(* POU Выборка значения из массива/Get_Speed_ARRAY_Number, ST *)
FUNCTION Get_Speed_ARRAY_Number : BYTE
VAR_INPUT
	Volume_now:DINT;
END_VAR
VAR
	i:BYTE:=1;
	j,ArraySize:BYTE:=12;
	med:BYTE;
END_VAR
(* Функция в качестве аргумента принимает, давление надува в мВольтах, а возвращает номер элемента массива, соответствующего этому количеству оборотов *)


(* Делим массив каждый раз пополам, проверяя где находится искомый элемент, пока границы массива не сойдутся*)

WHILE i<>j  DO
	med:=(i+j)/2;
	IF Volume_now > p.Speed_table[med] THEN
		i:=med+1;
	ELSE
		j:=med;
	END_IF
END_WHILE


Get_Speed_ARRAY_Number :=i;							(* Номер , когда границы сошлись и совпадают с краями массива не нуждается в уточнении *)

(* Уточняем какой элемент массива наиболее сответствует, кол-ву оборотов переданному как элемент функции *)
(* определяем спава или слева от найдено индекса находится ребуемый элемент и в зависмимости от этого действеум *)

IF i=med AND i<>1 THEN
	IF ABS(p.Speed_table[med-1]-Volume_now)<= ABS(p.Speed_table[med]-Volume_now) THEN
		Get_Speed_ARRAY_Number :=med-1;
	ELSE
		Get_Speed_ARRAY_Number :=med;
	END_IF
ELSIF i<>med AND  i<>ArraySize THEN
	IF ABS(p.Speed_table[med+1]-Volume_now)<= ABS(p.Speed_table[med]-Volume_now) THEN
		Get_Speed_ARRAY_Number :=med+1;
	ELSE
		Get_Speed_ARRAY_Number :=med;
	END_IF
END_IF
END_FUNCTION

(* POU Выборка значения из массива/Get_PPS_ARRAY_Number, ST *)
FUNCTION Get_PPS_ARRAY_Number : BYTE
VAR_INPUT
	PPS_now:DINT;
END_VAR
VAR
	i:BYTE:=1;
	j,ArraySize:BYTE:=32;
	med:BYTE;
END_VAR
(* Функция в качестве аргумента принимает, PPS, а возвращает номер элемента массива, соответствующего этому PPS *)

(* Делим массив каждый раз пополам, проверяя где находится искомый элемент, пока границы массива не сойдутся*)

WHILE i<>j  DO
	med:=(i+j)/2;
	IF PPS_now>p.PPS_table[med] THEN
		i:=med+1;
	ELSE
		j:=med;
	END_IF
END_WHILE


Get_PPS_ARRAY_Number :=i;							(* Номер , когда границы сошлись и совпадают с краями массива не нуждается в уточнении *)

(* Уточняем какой элемент массива наиболее сответствует, кол-ву оборотов переданному как элемент функции *)
(* определяем спава или слева от найдено индекса находится ребуемый элемент и в зависмимости от этого действеум *)

IF i=med AND i<>1 THEN
	IF ABS(p.PPS_table[med-1]-PPS_now)<= ABS(p.RPM_table[med]-PPS_now) THEN
		Get_PPS_ARRAY_Number :=med-1;
	ELSE
		Get_PPS_ARRAY_Number :=med;
	END_IF
ELSIF i<>med AND  i<>ArraySize THEN
	IF ABS(p.PPS_table[med+1]-PPS_now)<= ABS(p.PPS_table[med]-PPS_now) THEN
		Get_PPS_ARRAY_Number :=med+1;
	ELSE
		Get_PPS_ARRAY_Number :=med;
	END_IF
END_IF
END_FUNCTION

(* POU Ввод данных/Get_Turbo, ST *)
PROGRAM Get_Turbo
VAR
	s16_Return      : INT;
   fb_InGetValue   : FB_x_in_get_value;
END_VAR
fb_InGetValue(ou16_Channel:=X_IN_21, os32_Value=>Turbo_pressure, os16_Status=>s16_Return);
END_PROGRAM

(* POU Ввод данных/Get_Key, ST *)
PROGRAM Get_Key
VAR
	s16_Return      : INT;
   fb_InGetValue   : FB_x_in_get_value;

	DF_switch	:DINT;
	DF_flag		:BOOL;

END_VAR
fb_InGetValue(ou16_Channel:=X_IN_12, os32_Value=>DF_switch, os16_Status=>s16_Return);

IF DF_switch=0 THEN					(* Если конпока изменения режима работы ECU нажата, то...*)
	IF DF_flag THEN					(* Первый ли цикл когда она нажата ? *)
		DF_flag:=FALSE;				(*Выставляем флажок, для  игнорирования этой ветви, до тех пор пока кнопка не изменит своего положения *)
		IF Flag_ECU_ON THEN			(* Включаем или выключаем газодизельный режим ECU*)
			Flag_ECU_ON:=FALSE;
		ELSE
			Flag_ECU_ON:=TRUE;
			Count_min_reductor_press:=0; (* При переключении режимов начать отчет времени когда далвение было минимальным с 0 *)
		END_IF;
	END_IF
ELSE
	DF_flag:=TRUE;				(* Кнопка была отпущена, устанвкливаем разрешительный флажок для обработки следующего нажатия *)
END_IF
END_PROGRAM

(* POU Ввод данных/Get_Gas_meter, ST *)
PROGRAM Get_Gas_meter
VAR
	s16_Return      : INT;
   fb_InGetValue   : FB_x_in_get_value;
	fb_OutSetValue   : FB_x_out_set_value;

	i: DINT;
END_VAR
(* Считать значениедатчика кол-ва газа *)
fb_InGetValue(ou16_Channel:=X_IN_19, os32_Value=>Gas_meter, os16_Status=>s16_Return);

(* Определить уровень PWM для зажигания LED *)
i:=p.LED_BAR_PWM[Get_Gas_meter_ARRAY_Number(Gas_meter)];

(* Выдать PWM на LED bar *)
fb_OutSetValue(ou16_Channel:=X_OUT_03, os32_Value:=i, os16_Status=>s16_Return);
END_PROGRAM

(* POU Выборка значения из массива/Get_Gas_meter_ARRAY_Number, ST *)
FUNCTION Get_Gas_meter_ARRAY_Number : BYTE
VAR_INPUT
	Gas_meter_now:DINT;
END_VAR
VAR
	i:BYTE:=1;
	j,ArraySize:BYTE:=5;
	med:BYTE;

END_VAR
(* Функция в качестве аргумента принимает, количество оборотов, а возвращает номер элемента массива, соответствующего этому PPS *)


(* Делим массив каждый раз пополам, проверяя где находится искомый элемент, пока границы массива не сойдутся*)

WHILE i<>j  DO
	med:=(i+j)/2;
	IF Gas_meter_now>p.Gas_meter_volume[med] THEN
		i:=med+1;
	ELSE
		j:=med;
	END_IF
END_WHILE


Get_Gas_meter_ARRAY_Number :=i;							(* Номер , когда границы сошлись и совпадают с краями массива не нуждается в уточнении *)

(* Уточняем какой элемент массива наиболее сответствует, кол-ву оборотов переданному как элемент функции *)
(* определяем спава или слева от найдено индекса находится ребуемый элемент и в зависмимости от этого действеум *)

IF i=med AND i<>1 THEN
	IF ABS(p.Gas_meter_volume[med-1]-Gas_meter_now)<= ABS(p.Gas_meter_volume[med]-Gas_meter_now) THEN
		Get_Gas_meter_ARRAY_Number :=med-1;
	ELSE
		Get_Gas_meter_ARRAY_Number :=med;
	END_IF
ELSIF i<>med AND  i<>ArraySize THEN
	IF ABS(p.Gas_meter_volume[med+1]-Gas_meter_now)<= ABS(p.Gas_meter_volume[med]-Gas_meter_now) THEN
		Get_Gas_meter_ARRAY_Number :=med+1;
	ELSE
		Get_Gas_meter_ARRAY_Number :=med;
	END_IF
END_IF
END_FUNCTION

(* POU Ввод данных/Get_Reductor_temp, ST *)
PROGRAM Get_Reductor_temp
VAR
	s16_Return      : INT;
   fb_InGetValue   : FB_x_in_get_value;

	(* Температура редуктора уже в норме, время до следующей проверки пошло *)
	Flag_Err_Reductor_temp: BOOL;
	(* Счетчик циклов до следующей проверки *)
	Count_max_Reductor_temp: WORD;

END_VAR
fb_InGetValue(ou16_Channel:=X_IN_20, os32_Value=>Reductor_temp, os16_Status=>s16_Return);

(* Если температура редуктора превысила допустимую температуру для включения, то следующий
контроль произойдет через некоторое время,что бы избежать дребезга *)

IF Flag_Err_Reductor_temp AND  Count_max_Reductor_temp < Reductor_temp_err_time THEN
	Count_max_reductor_temp:=Count_max_reductor_temp+1;
ELSE
	Count_max_Reductor_temp:=0;
	(* Находится ли температура редуктора в допустимых пределах ? *)
	IF Reductor_temp < p.Reductor_temp_work THEN
		Flag_Err_Reductor_temp:=TRUE;
		Err_Reductor_temp:=TRUE;
	ELSE
		Flag_Err_Reductor_temp:=FALSE;
		Err_Reductor_temp:=FALSE;
	END_IF
END_IF
END_PROGRAM

(* POU Ввод данных/Get_Inj_temp, ST *)
PROGRAM Get_Inj_temp
VAR
	s16_Return      : INT;
   fb_InGetValue   : FB_x_in_get_value;
END_VAR
fb_InGetValue(ou16_Channel:=X_IN_15, os32_Value=>Injector_temp, os16_Status=>s16_Return);

(* Находится ли температура форсунок в допустимых пределах ? *)
(* Если температура форсунок хоть один раз превысила допустимый порог, то снять ошибку можно только перегрузкой *)

IF Injector_temp > p.Inj_temp_max THEN
	Err_inj_temp:=TRUE;
END_IF
END_PROGRAM

(* POU Ввод данных/Get_FUEL_meter, ST *)
PROGRAM Get_FUEL_meter
VAR
	s16_Return      : INT;
   fb_InGetValue   : FB_x_in_get_value;
	fb_OutSetValue   : FB_x_out_set_value;
	q: WORD;
END_VAR
(* Считать значениедатчика кол-ва солярки *)
fb_InGetValue(ou16_Channel:=X_IN_18, os32_Value=>FUEL_meter, os16_Status=>s16_Return);
(*Взять из таблицы физическое згачение объема слоответствующее показанию датчика *)
q:= p.FUEL_meter_liter[ Get_FUEL_meter_ARRAY_Number(FUEL_meter)];
FUEL_volume:=DINT_TO_REAL(FUEL_meter) * WORD_TO_REAL( q );
IF p.FUEL_meter_dat[Get_FUEL_meter_ARRAY_Number(FUEL_meter)] <> 0 THEN
	FUEL_volume:=FUEL_volume/WORD_TO_REAL(p.FUEL_meter_dat[Get_FUEL_meter_ARRAY_Number(FUEL_meter)]);
END_IF
END_PROGRAM

(* POU Выборка значения из массива/Get_FUEL_meter_ARRAY_Number, ST *)
FUNCTION Get_FUEL_meter_ARRAY_Number : BYTE
VAR_INPUT
	FUEL_meter_now:DINT;
END_VAR
VAR
	i:BYTE:=1;
	j,ArraySize:BYTE:=32;
	med:BYTE;

END_VAR
(* Функция в качестве аргумента принимает, количество оборотов, а возвращает номер элемента массива, соответствующего этому PPS *)


(* Делим массив каждый раз пополам, проверяя где находится искомый элемент, пока границы массива не сойдутся*)

WHILE i<>j  DO
	med:=(i+j)/2;
	IF FUEL_meter_now>p.FUEL_meter_dat[med] THEN
		i:=med+1;
	ELSE
		j:=med;
	END_IF
END_WHILE


Get_FUEL_meter_ARRAY_Number :=i;							(* Номер , когда границы сошлись и совпадают с краями массива не нуждается в уточнении *)

(* Уточняем какой элемент массива наиболее сответствует, кол-ву оборотов переданному как элемент функции *)
(* определяем спава или слева от найдено индекса находится ребуемый элемент и в зависмимости от этого действеум *)

IF i=med AND i<>1 THEN
	IF ABS(p.FUEL_meter_dat[med-1]-FUEL_meter_now)<= ABS(p.FUEL_meter_dat[med]-FUEL_meter_now) THEN
		Get_FUEL_meter_ARRAY_Number :=med-1;
	ELSE
		Get_FUEL_meter_ARRAY_Number :=med;
	END_IF
ELSIF i<>med AND  i<>ArraySize THEN
	IF ABS(p.FUEL_meter_dat[med+1]-FUEL_meter_now)<= ABS(p.FUEL_meter_dat[med]-FUEL_meter_now) THEN
		Get_FUEL_meter_ARRAY_Number :=med+1;
	ELSE
		Get_FUEL_meter_ARRAY_Number :=med;
	END_IF
END_IF
END_FUNCTION

(* POU Ввод данных/Get_cPPS, ST *)
PROGRAM Get_cPPS
VAR
	fb_InGetValue   : FB_x_in_get_value;
	s16_Return      : INT;
END_VAR
(* Взяьть реальное значение выдаваемого напряжения эмуляции PPS *)
fb_InGetValue(ou16_Channel:=X_IN_26, os32_Value=>cPPS1_emul, os16_Status=>s16_Return);
END_PROGRAM

(* POU CAN/Send, ST *)
PROGRAM Send
VAR
	s16_Return       		: INT;
	t_Msg             	: T_x_can_msg;
   fb_CanObjSendMsg   	: FB_x_can_obj_send_msg;
	fb_EepRead  			: FB_x_eep_read;
	u16_Crc           	: UINT;
	fb_UtiCalcCrc16   	: FB_x_uti_calc_crc_16;
	CAN_TX_count			:WORD:=10000;				(* Счетчик переданных пакетов по CAN *)

END_VAR
IF Flag_CAN THEN

	IF Flag_CAN_Write THEN
		Flag_CAN_Write:=FALSE;
		t_Msg.t_Id.u32_Id := 16#101;
		t_Msg.t_Id.u8_Xtd := 0;
		t_Msg.u8_Dlc      := 8;				(* Количество передаваемых байт *)
		t_Msg.au8_Data[0] := 1;
		t_Msg.au8_Data[1] := 9;
		t_Msg.au8_Data[2] := 7;
		t_Msg.au8_Data[3] := 2;
		t_Msg.au8_Data[4] := 1;
		t_Msg.au8_Data[5] := 9;
		t_Msg.au8_Data[6] := 7;
		t_Msg.au8_Data[7] := 2;
		fb_CanObjSendMsg(ou32_Handle:=TX, ot_Msg:=t_Msg, os16_Status=>s16_Return);
	END_IF


	IF Flag_CAN_send THEN											(* Первоначальная процедура, выполняется один раз по команде от Питоновской программе *)
		(* Читаем все содержимое энергонезависимой памяти *)
		fb_EepRead(ou32_Address:=0, ou32_Count:=SIZEOF(Can_buffer), opu8_Data:=ADR(Can_buffer), os16_Status=>s16_Return);
		(* Вычисляем CRC16 для массива передаваемых данных *)
		u16_Crc:=16#1D0F;
		fb_UtiCalcCrc16(ou32_Count:=SIZEOF(Can_buffer)-2, opu8_Data:=ADR(Can_buffer), ou16_Crc:=u16_Crc, os16_Status=>s16_Return);
		Can_buffer[SIZEOF(Can_buffer)-1]:=WORD_TO_BYTE(u16_Crc);
		Can_buffer[SIZEOF(Can_buffer)]:=WORD_TO_BYTE(u16_Crc/256);
		CAN_TX_count:=0;
		Flag_CAN_send:=FALSE;


	ELSIF CAN_TX_count <=  (SIZEOF(Can_buffer)-8) THEN						(* Передача основных данных, выполняется 1 раз после хандшейка *)

			(* Постоянная часть передачи *)
			t_Msg.t_Id.u32_Id := 16#101;		(* Адрес пакета *)
			t_Msg.t_Id.u8_Xtd := 0;
			t_Msg.u8_Dlc      := 8;				(* Количество передаваемых байт *)
			t_Msg.au8_Data[0] := Can_buffer[CAN_TX_count+1];
			t_Msg.au8_Data[1] := Can_buffer[CAN_TX_count+2];
			t_Msg.au8_Data[2] := Can_buffer[CAN_TX_count+3];
			t_Msg.au8_Data[3] := Can_buffer[CAN_TX_count+4];
			t_Msg.au8_Data[4] := Can_buffer[CAN_TX_count+5];
			t_Msg.au8_Data[5] := Can_buffer[CAN_TX_count+6];
			t_Msg.au8_Data[6] := Can_buffer[CAN_TX_count+7];
			t_Msg.au8_Data[7] := Can_buffer[CAN_TX_count+8];
			fb_CanObjSendMsg(ou32_Handle:=TX, ot_Msg:=t_Msg, os16_Status=>s16_Return);
			CAN_TX_count:=CAN_TX_count+8;
		END_IF

END_IF
END_PROGRAM

(* POU CAN/Recieve, ST *)
PROGRAM Recieve
VAR
	s16_Return        	: INT;
	r_Msg			         : T_x_can_msg;
	fb_CanObjGetMsg   	: FB_x_can_obj_get_msg;
	fb_EepWrite  			: FB_x_eep_write;

	u16_Crc           	: UINT;
	fb_UtiCalcCrc16   	: FB_x_uti_calc_crc_16;
	i: WORD; (* Счетчик принятых по CAN пакетов в калибровке *)

	crc_given: UINT;
END_VAR
IF Flag_CAN THEN
			(* Что бы при ошибке чтения с CANa , при не изменении значений не произошо ложного срабатывания *)
			r_Msg.au8_Data[0]:=0;r_Msg.au8_Data[1]:=0;r_Msg.au8_Data[2]:=0;r_Msg.au8_Data[3]:=0;r_Msg.au8_Data[4]:=0;
			r_Msg.au8_Data[5]:=0;r_Msg.au8_Data[6]:=0;r_Msg.au8_Data[7]:=0;
			fb_CanObjGetMsg(ou32_Handle:=RX, ot_Msg=>r_Msg, os16_Status=>s16_Return);
			IF s16_Return = C_NO_ERR THEN

					(* Поступил запрос на передачу? *)
					IF	Flag_CAN_recieve=FALSE AND r_Msg.au8_Data[0] = 8 AND r_Msg.au8_Data[1] = 7 AND r_Msg.au8_Data[2] = 6 AND r_Msg.au8_Data[3] = 5 AND
						r_Msg.au8_Data[4] = 4 AND r_Msg.au8_Data[5] = 3 AND r_Msg.au8_Data[6] = 2 AND	r_Msg.au8_Data[7] = 1 THEN
						Flag_CAN_send:=TRUE;
					END_IF

					(* Поступил запрос на прием ? *)
					IF Flag_CAN_recieve = FALSE AND r_Msg.au8_Data[0] = 1 AND r_Msg.au8_Data[1] = 2 AND r_Msg.au8_Data[2] = 3 AND r_Msg.au8_Data[3] = 4 AND
						r_Msg.au8_Data[4] = 5 AND r_Msg.au8_Data[5] = 6 AND r_Msg.au8_Data[6] = 7 AND r_Msg.au8_Data[7] = 8 THEN

									Flag_CAN_recieve:=TRUE;
									i:=1;
					ELSIF i <= SIZEOF(Can_buffer)-7 THEN
											Can_buffer[i]:=r_Msg.au8_Data[0]; Can_buffer[i+1]:=r_Msg.au8_Data[1]; Can_buffer[i+2]:=r_Msg.au8_Data[2]; Can_buffer[i+3]:=r_Msg.au8_Data[3];
											Can_buffer[i+4]:=r_Msg.au8_Data[4]; Can_buffer[i+5]:=r_Msg.au8_Data[5]; Can_buffer[i+6]:=r_Msg.au8_Data[6]; Can_buffer[i+7]:=r_Msg.au8_Data[7];
											i:=i+8;
											IF i=SIZEOF(Can_buffer)+1 THEN
													Flag_CAN_recieve:= FALSE;
													(* Вычисляем CRC16 для массива передаваемых данных *)
													u16_Crc:=16#1D0F;
													fb_UtiCalcCrc16(ou32_Count:=SIZEOF(Can_buffer)-2, opu8_Data:=ADR(Can_buffer), ou16_Crc:=u16_Crc, os16_Status=>s16_Return);
													crc_given:= Can_buffer[SIZEOF(Can_buffer)]*256+Can_buffer[SIZEOF(Can_buffer)-1];
													IF crc_given =  u16_Crc THEN
															fb_EepWrite(ou32_Address:=0, ou32_Count:=SIZEOF(Can_buffer), opu8_Data:=ADR(Can_buffer), os16_Status=>s16_Return);
															Flag_CAN_Write:= TRUE;
													END_IF
											END_IF
					END_IF

			END_IF
END_IF
END_PROGRAM

(* Visualisation CALIBRATION
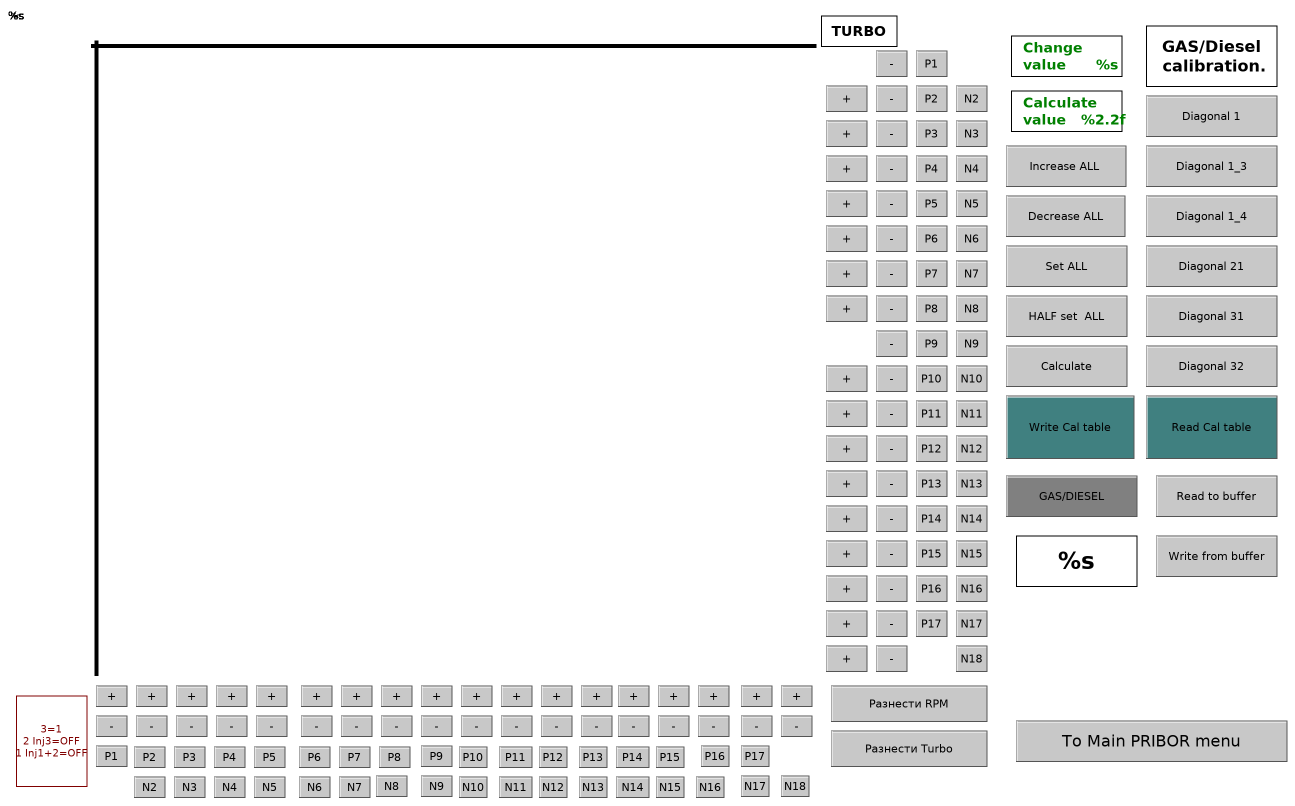
rectangle at (0,0)-(0,0): text "%s"; shows p.RPM_table[INDEX]; editable
rectangle at (0,0)-(0,0): text "%s"; shows p.Turbo_table[1]; editable
rectangle at (0,0)-(0,0): text "%s"; shows p.Turbo_table[2]; editable
rectangle at (0,0)-(0,0): text "%s"; shows p.Turbo_table[3]; editable
rectangle at (0,0)-(0,0): text "%s"; shows p.Turbo_table[4]; editable
rectangle at (0,0)-(0,0): text "%s"; shows p.Turbo_table[5]; editable
rectangle at (0,0)-(0,0): text "%s"; shows p.Turbo_table[6]; editable
rectangle at (0,0)-(0,0): text "%s"; shows p.Turbo_table[7]; editable
rectangle at (0,0)-(0,0): text "%s"; shows p.Turbo_table[8]; editable
rectangle at (0,0)-(0,0): text "%s"; shows p.Turbo_table[9]; editable
rectangle at (0,0)-(0,0): text "%s"; shows p.Turbo_table[10]; editable
rectangle at (0,0)-(0,0): text "%s"; shows p.Turbo_table[11]; editable
rectangle at (0,0)-(0,0): text "%s"; shows p.Turbo_table[12]; editable
rectangle at (0,0)-(0,0): text "%s"; shows p.Turbo_table[13]; editable
rectangle at (0,0)-(0,0): text "%s"; shows p.Turbo_table[14]; editable
rectangle at (0,0)-(0,0): text "%s"; shows p.Turbo_table[15]; editable
rectangle at (0,0)-(0,0): text "%s"; shows p.Turbo_table[16]; editable
rectangle at (0,0)-(0,0): text "%s"; shows p.Turbo_table[17]; editable
rectangle at (0,0)-(0,0): text "%s"; shows p.Turbo_table[18]; editable
button at (990,130)-(1110,171): text "Increase ALL"; taps DFPRS_Change_Cal_Table.ALL_plus
button at (990,180)-(1109,221): text "Decrease ALL"; taps DFPRS_Change_Cal_Table.ALL_minus
button at (1130,380)-(1261,443): text "Read Cal table"; taps DFPRS_Change_Cal_Table.Read_cal
button at (990,380)-(1118,443): text "Write Cal table"; taps DFPRS_Change_Cal_Table.Write_cal
button at (990,230)-(1111,271): text "Set ALL"; taps DFPRS_Change_Cal_Table.Set_ALL
button at (990,280)-(1111,321): text "HALF set  ALL"; taps DFPRS_Change_Cal_Table.HALF_set_ALL
button at (860,35)-(891,61): text "-"; taps DFPRS_Change_Cal_Table.RPM_Flag_minus_1
button at (810,70)-(851,96): text "+"; taps DFPRS_Change_Cal_Table.RPM_Flag_plus_2
button at (860,70)-(891,96): text "-"; taps DFPRS_Change_Cal_Table.RPM_Flag_minus_2
button at (900,70)-(931,96): text "P2"; taps DFPRS_Change_Cal_Table.RPM_Flag_CP_2
button at (810,105)-(851,131): text "+"; taps DFPRS_Change_Cal_Table.RPM_Flag_plus_3
button at (860,105)-(891,131): text "-"; taps DFPRS_Change_Cal_Table.RPM_Flag_minus_3
button at (900,105)-(931,131): text "P3"; taps DFPRS_Change_Cal_Table.RPM_Flag_CP_3
button at (810,140)-(851,166): text "+"; taps DFPRS_Change_Cal_Table.RPM_Flag_plus_4
button at (860,140)-(891,166): text "-"; taps DFPRS_Change_Cal_Table.RPM_Flag_minus_4
button at (900,140)-(931,166): text "P4"; taps DFPRS_Change_Cal_Table.RPM_Flag_CP_4
button at (810,175)-(851,201): text "+"; taps DFPRS_Change_Cal_Table.RPM_Flag_plus_5
button at (860,175)-(891,201): text "-"; taps DFPRS_Change_Cal_Table.RPM_Flag_minus_5
button at (900,175)-(931,201): text "P5"; taps DFPRS_Change_Cal_Table.RPM_Flag_CP_5
button at (810,210)-(851,236): text "+"; taps DFPRS_Change_Cal_Table.RPM_Flag_plus_6
button at (860,210)-(891,236): text "-"; taps DFPRS_Change_Cal_Table.RPM_Flag_minus_6
button at (900,210)-(931,236): text "P6"; taps DFPRS_Change_Cal_Table.RPM_Flag_CP_6
button at (810,245)-(851,271): text "+"; taps DFPRS_Change_Cal_Table.RPM_Flag_plus_7
button at (860,245)-(891,271): text "-"; taps DFPRS_Change_Cal_Table.RPM_Flag_minus_7
button at (900,245)-(931,271): text "P7"; taps DFPRS_Change_Cal_Table.RPM_Flag_CP_7
button at (810,280)-(851,306): text "+"; taps DFPRS_Change_Cal_Table.RPM_Flag_plus_8
button at (860,280)-(891,306): text "-"; taps DFPRS_Change_Cal_Table.RPM_Flag_minus_8
button at (900,280)-(931,306): text "P8"; taps DFPRS_Change_Cal_Table.RPM_Flag_CP_8
button at (80,670)-(111,691): text "+"; taps DFPRS_Change_Cal_Table.Turbo_Flag_plus_1
button at (80,700)-(111,721): text "-"; taps DFPRS_Change_Cal_Table.Turbo_Flag_minus_1
button at (120,670)-(151,691): text "+"; taps DFPRS_Change_Cal_Table.Turbo_Flag_plus_2
button at (120,700)-(151,721): text "-"; taps DFPRS_Change_Cal_Table.Turbo_Flag_minus_2
button at (118,731)-(149,752): text "P2"; taps DFPRS_Change_Cal_Table.Turbo_Flag_CP_2
button at (160,670)-(191,691): text "+"; taps DFPRS_Change_Cal_Table.Turbo_Flag_plus_3
button at (160,700)-(191,721): text "-"; taps DFPRS_Change_Cal_Table.Turbo_Flag_minus_3
button at (158,731)-(189,752): text "P3"; taps DFPRS_Change_Cal_Table.Turbo_Flag_CP_3
button at (200,670)-(231,691): text "+"; taps DFPRS_Change_Cal_Table.Turbo_Flag_plus_4
button at (200,700)-(231,721): text "-"; taps DFPRS_Change_Cal_Table.Turbo_Flag_minus_4
button at (198,731)-(229,752): text "P4"; taps DFPRS_Change_Cal_Table.Turbo_Flag_CP_4
button at (240,670)-(271,691): text "+"; taps DFPRS_Change_Cal_Table.Turbo_Flag_plus_5
button at (240,700)-(271,721): text "-"; taps DFPRS_Change_Cal_Table.Turbo_Flag_minus_5
button at (238,731)-(269,752): text "P5"; taps DFPRS_Change_Cal_Table.Turbo_Flag_CP_5
button at (285,670)-(316,691): text "+"; taps DFPRS_Change_Cal_Table.Turbo_Flag_plus_6
button at (285,700)-(316,721): text "-"; taps DFPRS_Change_Cal_Table.Turbo_Flag_minus_6
button at (283,731)-(314,752): text "P6"; taps DFPRS_Change_Cal_Table.Turbo_Flag_CP_6
button at (325,670)-(356,691): text "+"; taps DFPRS_Change_Cal_Table.Turbo_Flag_plus_7
button at (325,700)-(356,721): text "-"; taps DFPRS_Change_Cal_Table.Turbo_Flag_minus_7
button at (323,731)-(354,752): text "P7"; taps DFPRS_Change_Cal_Table.Turbo_Flag_CP_7
button at (365,670)-(396,691): text "+"; taps DFPRS_Change_Cal_Table.Turbo_Flag_plus_8
button at (365,700)-(396,721): text "-"; taps DFPRS_Change_Cal_Table.Turbo_Flag_minus_8
button at (363,731)-(394,752): text "P8"; taps DFPRS_Change_Cal_Table.Turbo_Flag_CP_8
rounded rectangle at (995,20)-(1106,61): text "Change / value      %s"; shows DFPRS_Change_Cal_Table.Change_volume; editable 0..
rounded rectangle at (1130,10)-(1261,71): text "GAS/Diesel / calibration."
button at (1140,460)-(1261,501): text "Read to buffer"; taps DFPRS_Change_Cal_Table.red_cal2
button at (1140,520)-(1261,561): text "Write from buffer"; taps DFPRS_Change_Cal_Table.Write_cal2
button at (860,315)-(891,341): text "-"; taps DFPRS_Change_Cal_Table.RPM_Flag_minus_9
button at (810,350)-(851,376): text "+"; taps DFPRS_Change_Cal_Table.RPM_Flag_plus_10
button at (860,350)-(891,376): text "-"; taps DFPRS_Change_Cal_Table.RPM_Flag_minus_10
button at (900,350)-(931,376): text "P10"; taps DFPRS_Change_Cal_Table.RPM_Flag_CP_10
button at (810,385)-(851,411): text "+"; taps DFPRS_Change_Cal_Table.RPM_Flag_plus_11
button at (860,385)-(891,411): text "-"; taps DFPRS_Change_Cal_Table.RPM_Flag_minus_11
button at (900,385)-(931,411): text "P11"; taps DFPRS_Change_Cal_Table.RPM_Flag_CP_11
button at (810,420)-(851,446): text "+"; taps DFPRS_Change_Cal_Table.RPM_Flag_plus_12
button at (860,420)-(891,446): text "-"; taps DFPRS_Change_Cal_Table.RPM_Flag_minus_12
button at (900,420)-(931,446): text "P12"; taps DFPRS_Change_Cal_Table.RPM_Flag_CP_12
button at (810,455)-(851,481): text "+"; taps DFPRS_Change_Cal_Table.RPM_Flag_plus_13
button at (860,455)-(891,481): text "-"; taps DFPRS_Change_Cal_Table.RPM_Flag_minus_13
button at (900,455)-(931,481): text "P13"; taps DFPRS_Change_Cal_Table.RPM_Flag_CP_13
button at (900,315)-(931,341): text "P9"; taps DFPRS_Change_Cal_Table.RPM_Flag_CP_9
button at (405,670)-(436,691): text "+"; taps DFPRS_Change_Cal_Table.Turbo_Flag_plus_9
button at (405,700)-(436,721): text "-"; taps DFPRS_Change_Cal_Table.Turbo_Flag_minus_9
button at (445,670)-(476,691): text "+"; taps DFPRS_Change_Cal_Table.Turbo_Flag_plus_10
button at (445,700)-(476,721): text "-"; taps DFPRS_Change_Cal_Table.Turbo_Flag_minus_10
button at (443,731)-(471,752): text "P10"; taps DFPRS_Change_Cal_Table.Turbo_Flag_CP_10
button at (485,670)-(516,691): text "+"; taps DFPRS_Change_Cal_Table.Turbo_Flag_plus_11
button at (485,700)-(516,721): text "-"; taps DFPRS_Change_Cal_Table.Turbo_Flag_minus_11
button at (483,731)-(516,752): text "P11"; taps DFPRS_Change_Cal_Table.Turbo_Flag_CP_11
button at (525,670)-(556,691): text "+"; taps DFPRS_Change_Cal_Table.Turbo_Flag_plus_12
button at (525,700)-(556,721): text "-"; taps DFPRS_Change_Cal_Table.Turbo_Flag_minus_12
button at (523,731)-(551,752): text "P12"; taps DFPRS_Change_Cal_Table.Turbo_Flag_CP_12
button at (565,670)-(596,691): text "+"; taps DFPRS_Change_Cal_Table.Turbo_Flag_plus_13
button at (565,700)-(596,721): text "-"; taps DFPRS_Change_Cal_Table.Turbo_Flag_minus_13
button at (563,731)-(591,752): text "P13"; taps DFPRS_Change_Cal_Table.Turbo_Flag_CP_13
button at (405,730)-(436,751): text "P9"; taps DFPRS_Change_Cal_Table.Turbo_Flag_CP_9
rectangle at (0,680)-(71,771): text "3=1 / 2 Inj3=OFF / 1 Inj1+2=OFF"
button at (990,460)-(1121,501): text "GAS/DIESEL"; toggles DFPRS_Change_Cal_Table.Flag_cal_table_gas
rounded rectangle at (1000,520)-(1121,571): text "%s"; shows DFPRS_Change_Cal_Table.Fuel_type
button at (990,330)-(1111,371): text "Calculate"; taps DFPRS_Change_Cal_Table.Calculate
rounded rectangle at (995,75)-(1106,116): text "Calculate / value   %2.2f"; shows .p.Calculate_volume; editable 0..
button at (1130,80)-(1261,121): text "Diagonal 1"; taps DFPRS_Change_Cal_Table.Diagonal_1
button at (810,490)-(851,516): text "+"; taps DFPRS_Change_Cal_Table.RPM_Flag_plus_14
button at (860,490)-(891,516): text "-"; taps DFPRS_Change_Cal_Table.RPM_Flag_minus_14
button at (900,490)-(931,516): text "P14"; taps DFPRS_Change_Cal_Table.RPM_Flag_CP_14
button at (810,525)-(851,551): text "+"; taps DFPRS_Change_Cal_Table.RPM_Flag_plus_15
button at (860,525)-(891,551): text "-"; taps DFPRS_Change_Cal_Table.RPM_Flag_minus_15
button at (900,525)-(931,551): text "P15"; taps DFPRS_Change_Cal_Table.RPM_Flag_CP_15
button at (810,560)-(851,586): text "+"; taps DFPRS_Change_Cal_Table.RPM_Flag_plus_16
button at (860,560)-(891,586): text "-"; taps DFPRS_Change_Cal_Table.RPM_Flag_minus_16
button at (900,35)-(931,61): text "P1"; taps DFPRS_Change_Cal_Table.RPM_Flag_CP_1
button at (940,70)-(971,96): text "N2"; taps DFPRS_Change_Cal_Table.RPM_Flag_CN_2
button at (940,105)-(971,131): text "N3"; taps DFPRS_Change_Cal_Table.RPM_Flag_CN_3
button at (940,140)-(971,166): text "N4"; taps DFPRS_Change_Cal_Table.RPM_Flag_CN_4
button at (940,175)-(971,201): text "N5"; taps DFPRS_Change_Cal_Table.RPM_Flag_CN_5
button at (940,210)-(971,236): text "N6"; taps DFPRS_Change_Cal_Table.RPM_Flag_CN_6
button at (940,245)-(971,271): text "N7"; taps DFPRS_Change_Cal_Table.RPM_Flag_CN_7
button at (940,280)-(971,306): text "N8"; taps DFPRS_Change_Cal_Table.RPM_Flag_CN_8
button at (940,350)-(971,376): text "N10"; taps DFPRS_Change_Cal_Table.RPM_Flag_CN_10
button at (940,385)-(971,411): text "N11"; taps DFPRS_Change_Cal_Table.RPM_Flag_CN_11
button at (940,420)-(971,446): text "N12"; taps DFPRS_Change_Cal_Table.RPM_Flag_CN_12
button at (940,455)-(971,481): text "N13"; taps DFPRS_Change_Cal_Table.RPM_Flag_CN_13
button at (940,315)-(971,341): text "N9"; taps DFPRS_Change_Cal_Table.RPM_Flag_CN_9
button at (940,490)-(971,516): text "N14"; taps DFPRS_Change_Cal_Table.RPM_Flag_CN_14
button at (940,525)-(971,551): text "N15"; taps DFPRS_Change_Cal_Table.RPM_Flag_CN_15
button at (940,560)-(971,586): text "N16"; taps DFPRS_Change_Cal_Table.RPM_Flag_CN_16
button at (1130,180)-(1261,221): text "Diagonal 1_4"; taps DFPRS_Change_Cal_Table.Diagonal_14
button at (1130,130)-(1261,171): text "Diagonal 1_3"; taps DFPRS_Change_Cal_Table.Diagonal_13
button at (1130,230)-(1261,271): text "Diagonal 21"; taps DFPRS_Change_Cal_Table.Diagonal_21
button at (1130,280)-(1261,321): text "Diagonal 31"; taps DFPRS_Change_Cal_Table.Diagonal_31
button at (1000,705)-(1271,746): text "To Main PRIBOR menu"; opens PLC_VISU
button at (602,670)-(633,691): text "+"; taps DFPRS_Change_Cal_Table.Turbo_Flag_plus_14
button at (602,700)-(633,721): text "-"; taps DFPRS_Change_Cal_Table.Turbo_Flag_minus_14
button at (600,731)-(633,752): text "P14"; taps DFPRS_Change_Cal_Table.Turbo_Flag_CP_14
button at (642,670)-(673,691): text "+"; taps DFPRS_Change_Cal_Table.Turbo_Flag_plus_15
button at (642,700)-(673,721): text "-"; taps DFPRS_Change_Cal_Table.Turbo_Flag_minus_15
button at (640,731)-(668,752): text "P15"; taps DFPRS_Change_Cal_Table.Turbo_Flag_CP_15
button at (682,670)-(713,691): text "+"; taps DFPRS_Change_Cal_Table.Turbo_Flag_plus_16
button at (682,700)-(713,721): text "-"; taps DFPRS_Change_Cal_Table.Turbo_Flag_minus_16
button at (80,730)-(111,751): text "P1"; taps DFPRS_Change_Cal_Table.Turbo_Flag_CP_1
button at (118,761)-(149,782): text "N2"; taps DFPRS_Change_Cal_Table.Turbo_Flag_CN_2
button at (158,761)-(189,782): text "N3"; taps DFPRS_Change_Cal_Table.Turbo_Flag_CN_3
button at (198,761)-(229,782): text "N4"; taps DFPRS_Change_Cal_Table.Turbo_Flag_CN_4
button at (238,761)-(269,782): text "N5"; taps DFPRS_Change_Cal_Table.Turbo_Flag_CN_5
button at (283,761)-(314,782): text "N6"; taps DFPRS_Change_Cal_Table.Turbo_Flag_CN_6
button at (323,761)-(354,782): text "N7"; taps DFPRS_Change_Cal_Table.Turbo_Flag_CN_7
button at (360,760)-(391,781): text "N8"; taps DFPRS_Change_Cal_Table.Turbo_Flag_CN_8
button at (443,761)-(471,782): text "N10"; taps DFPRS_Change_Cal_Table.Turbo_Flag_CN_10
button at (483,761)-(516,782): text "N11"; taps DFPRS_Change_Cal_Table.Turbo_Flag_CN_11
button at (523,761)-(551,782): text "N12"; taps DFPRS_Change_Cal_Table.Turbo_Flag_CN_12
button at (563,761)-(591,782): text "N13"; taps DFPRS_Change_Cal_Table.Turbo_Flag_CN_13
button at (405,760)-(436,781): text "N9"; taps DFPRS_Change_Cal_Table.Turbo_Flag_CN_9
button at (600,761)-(633,782): text "N14"; taps DFPRS_Change_Cal_Table.Turbo_Flag_CN_14
button at (640,761)-(668,782): text "N15"; taps DFPRS_Change_Cal_Table.Turbo_Flag_CN_15
button at (680,761)-(708,782): text "N16"; taps DFPRS_Change_Cal_Table.Turbo_Flag_CN_16
button at (1130,330)-(1261,371): text "Diagonal 32"; taps DFPRS_Change_Cal_Table.Diagonal_32
rectangle at (805,0)-(881,31): text "TURBO"
button at (810,595)-(851,621): text "+"; taps DFPRS_Change_Cal_Table.RPM_Flag_plus_17
button at (860,595)-(891,621): text "-"; taps DFPRS_Change_Cal_Table.RPM_Flag_minus_17
button at (810,630)-(851,656): text "+"; taps DFPRS_Change_Cal_Table.RPM_Flag_plus_18
button at (860,630)-(891,656): text "-"; taps DFPRS_Change_Cal_Table.RPM_Flag_minus_18
button at (725,670)-(756,691): text "+"; taps DFPRS_Change_Cal_Table.Turbo_Flag_plus_17
button at (725,700)-(756,721): text "-"; taps DFPRS_Change_Cal_Table.Turbo_Flag_minus_17
button at (765,670)-(796,691): text "+"; taps DFPRS_Change_Cal_Table.Turbo_Flag_plus_18
button at (765,700)-(796,721): text "-"; taps DFPRS_Change_Cal_Table.Turbo_Flag_minus_18
button at (900,595)-(931,621): text "P17"; taps DFPRS_Change_Cal_Table.RPM_Flag_CP_17
button at (940,595)-(971,621): text "N17"; taps DFPRS_Change_Cal_Table.RPM_Flag_CN_17
button at (940,630)-(971,656): text "N18"; taps DFPRS_Change_Cal_Table.RPM_Flag_CN_18
button at (900,560)-(931,586): text "P16"; taps DFPRS_Change_Cal_Table.RPM_Flag_CP_16
button at (725,730)-(753,751): text "P17"; taps DFPRS_Change_Cal_Table.Turbo_Flag_CP_17
button at (725,760)-(753,781): text "N17"; taps DFPRS_Change_Cal_Table.Turbo_Flag_CN_17
button at (765,760)-(793,781): text "N18"; taps DFPRS_Change_Cal_Table.Turbo_Flag_CN_18
button at (685,730)-(713,751): text "P16"; taps DFPRS_Change_Cal_Table.Turbo_Flag_CP_16
button at (815,670)-(971,706): text "Разнести RPM"; taps DFPRS_Change_Cal_Table.Flag_RPM_raznoska
button at (815,715)-(971,751): text "Разнести Turbo"; taps DFPRS_Change_Cal_Table.Flag_Turbo_raznoska
2 more shapes without text or variables
*)

(* Visualisation Check_parameters/CHECK_CURRENT
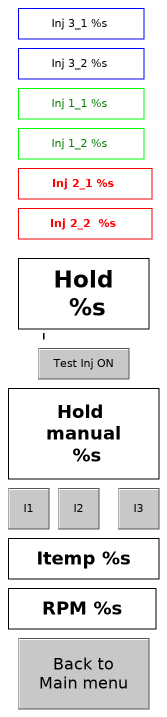
rounded rectangle at (1210,90)-(1336,121): text "Inj 1_1 %s"; shows .s32_Current_Inj1_1/1000
rounded rectangle at (1210,210)-(1344,241): text "Inj 2_2  %s"; shows .s32_Current_Inj2_2/1000
rounded rectangle at (1210,260)-(1341,331): text "Hold / %s"; shows .HOLD_time
rounded rectangle at (1210,10)-(1336,41): text "Inj 3_1 %s"; shows .s32_Current_Inj3_1/1000
rounded rectangle at (1210,130)-(1336,161): text "Inj 1_2 %s"; shows .s32_Current_Inj1_2/1000
rounded rectangle at (1210,170)-(1344,201): text "Inj 2_1 %s"; shows .s32_Current_Inj2_1/1000
rounded rectangle at (1210,50)-(1336,81): text "Inj 3_2 %s"; shows s32_Current_Inj3_2/1000
button at (1230,350)-(1321,381): text "Test Inj ON"; toggles .Flag_test_inj
rectangle at (1200,390)-(1351,481): text "Hold / manual / %s"; shows Act_control.Hold_manual; editable
button at (1200,490)-(1241,531): text "I1"; toggles .Flag_Inj1_ON
button at (1250,490)-(1291,531): text "I2"; toggles .Flag_Inj2_ON
button at (1310,490)-(1351,531): text "I3"; toggles .Flag_Inj3_ON
rounded rectangle at (1200,540)-(1351,581): text "Itemp %s"; shows .Injector_temp
rounded rectangle at (1200,590)-(1348,631): text "RPM %s"; shows .RPM
button at (1210,640)-(1341,711): text "Back to / Main menu"; opens PLC_VISU
1 more shapes without text or variables
1 elements of other kinds (tables, trends, ...) not read
*)

(* Visualisation Check_parameters/CHECK_EGT
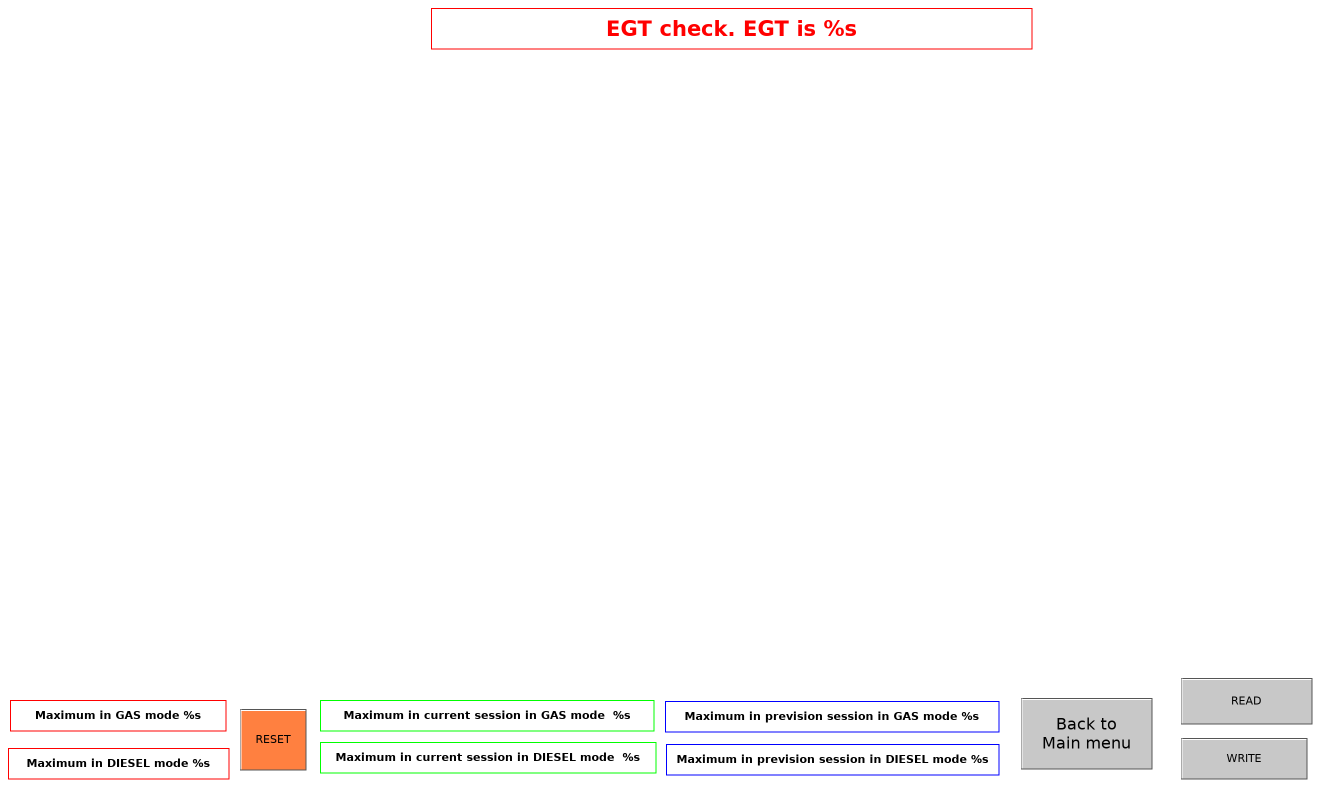
rounded rectangle at (9,702)-(225,733): text "Maximum in GAS mode %s"; shows .a.EGT_max_abs_GAS
rounded rectangle at (7,750)-(228,781): text "Maximum in DIESEL mode %s"; shows .a.EGT_max_abs_DIESEL
rounded rectangle at (665,746)-(998,777): text "Maximum in prevision session in DIESEL mode %s"; shows PLC_PRG.EGT_max_prev_sessions_DIESEL
rounded rectangle at (664,703)-(998,734): text "Maximum in prevision session in GAS mode %s"; shows PLC_PRG.EGT_max_prev_sessions_GAS
rounded rectangle at (319,702)-(653,733): text "Maximum in current session in GAS mode  %s"; shows .a.EGT_max_sessions_GAS
rounded rectangle at (319,744)-(655,775): text "Maximum in current session in DIESEL mode  %s"; shows .a.EGT_max_sessions_DIESEL
rounded rectangle at (430,10)-(1031,51): text "EGT check. EGT is %s"; shows .EGT
button at (239,711)-(305,772): text "RESET"; taps Get_EGT.Flag_EGT_reset
button at (1020,700)-(1151,771): text "Back to / Main menu"; opens PLC_VISU
button at (1180,680)-(1311,726): text "READ"; taps DFPRS_Change_Cal_Table.Read_cal
button at (1180,740)-(1306,781): text "WRITE"; taps DFPRS_Change_Cal_Table.Write_cal
1 elements of other kinds (tables, trends, ...) not read
*)

(* Visualisation PLC_VISU
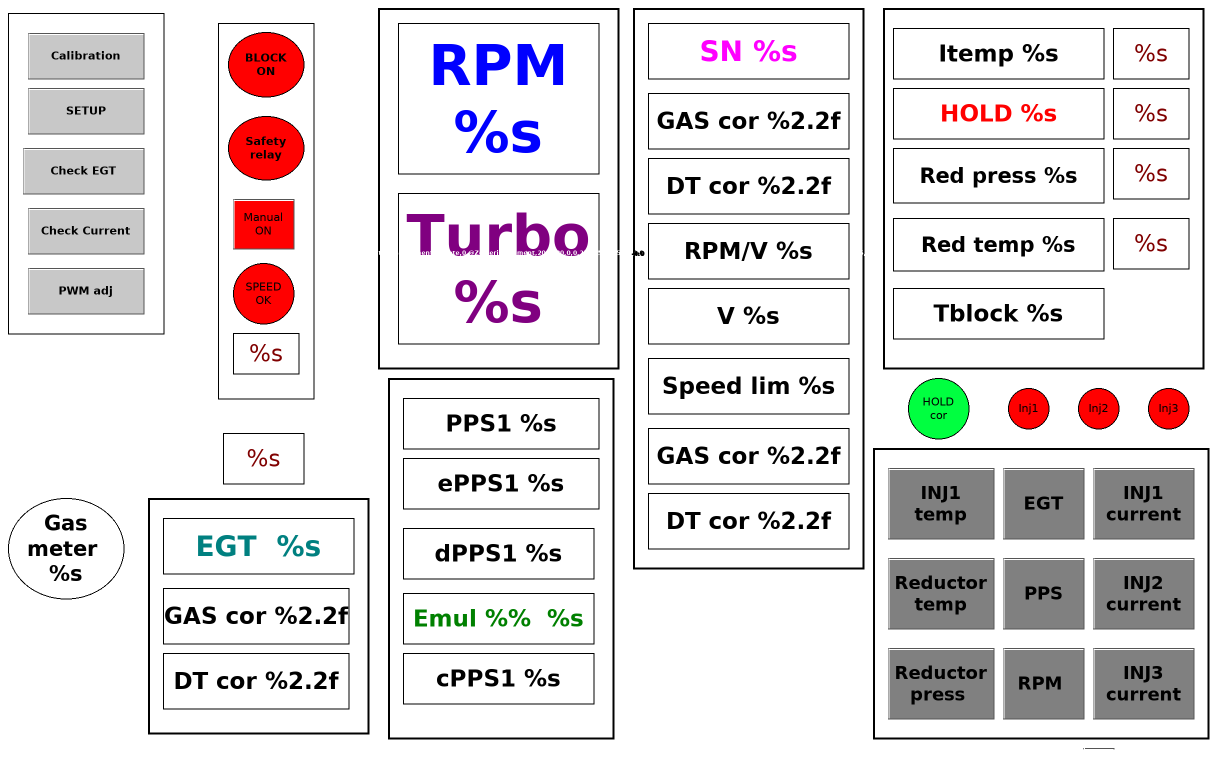
button at (1015,650)-(1096,721): text "RPM"; toggles .Err_RPM
button at (1015,470)-(1096,541): text "EGT"; toggles .Err_EGT
button at (900,560)-(1006,631): text "Reductor / temp"; toggles .Err_Reductor_temp
button at (900,650)-(1006,721): text "Reductor / press"; shows .Reductor_press; toggles .Err_Reductor_press
button at (1105,470)-(1206,541): text "INJ1 / current"; toggles .Err_Inj1
button at (1105,560)-(1206,631): text "INJ2 / current"; toggles .Err_Inj2
button at (900,470)-(1006,541): text "INJ1 / temp"; toggles .Err_Inj_temp
button at (1015,560)-(1096,631): text "PPS"; toggles .Err_PPS
button at (1105,650)-(1206,721): text "INJ3 / current"; toggles .Err_Inj3
ellipse at (1020,390)-(1061,431): text "Inj1"; alarm colour if .Flag_Inj1_ON
ellipse at (1090,390)-(1131,431): text "Inj2"; alarm colour if .Flag_Inj2_ON
ellipse at (1160,390)-(1201,431): text "Inj3"; alarm colour if .Flag_Inj3_ON
ellipse at (920,380)-(981,441): text "HOLD / cor"; alarm colour if .Flag_Inj_PWM_cor
group at (390,10)-(631,371)
  group at (10,210)-(11,211)
    rectangle at (0,0)-(1,1): text "{ExtendedElement},Visu\ElementDLL.ete,0,@Zeigerinstrument,200,180,0,0,255,255,255,0,,,%.1f,0,1,1,1,2,-4,4,0,0,0,0,0,0,0,-13,16,700,Arial,1,2,4000,5500,255,255,128,5500,6000,255,0,0,"
    rectangle at (1,92)-(23,108): text "-4.0"
    rectangle at (27,30)-(49,46): text "-2.0"
    rectangle at (91,4)-(109,20): text "0.0"
    rectangle at (153,30)-(171,46): text "2.0"
    rectangle at (179,92)-(197,108): text "4.0"
  rounded rectangle at (20,185)-(221,336): text "Turbo / %s"; shows .Turbo_pressure
  rounded rectangle at (20,15)-(221,166): text "RPM / %s"; shows .RPM
group at (650,255)-(651,256)
  rectangle at (0,0)-(1,1): text "{ExtendedElement},Visu\ElementDLL.ete,0,@Zeigerinstrument,200,180,0,0,255,255,255,0,,,%.1f,0,1,1,1,2,-4,4,0,0,0,0,0,0,0,-13,16,700,Arial,1,2,4000,5500,255,255,128,5500,6000,255,0,0,"
  rectangle at (1,92)-(23,108): text "-4.0"
  rectangle at (27,30)-(49,46): text "-2.0"
  rectangle at (91,4)-(109,20): text "0.0"
  rectangle at (153,30)-(171,46): text "2.0"
  rectangle at (179,92)-(197,108): text "4.0"
rounded rectangle at (660,225)-(861,281): text "RPM/V %s"; shows .Load
rounded rectangle at (660,290)-(861,346): text "V %s"; shows .Speed
rounded rectangle at (660,25)-(861,81): text "SN %s"; shows .Speed_number
rounded rectangle at (660,95)-(861,151): text "GAS cor %2.2f"; shows Act_control.Gas_cor
rounded rectangle at (660,160)-(861,216): text "DT cor %2.2f"; shows Act_control.Diesel_cor
ellipse at (20,500)-(136,601): text "Gas / meter / %s"; shows .Gas_meter
group at (400,380)-(626,741)
  rounded rectangle at (15,20)-(211,71): text "PPS1 %s"; shows .PPS1
  rounded rectangle at (15,80)-(211,131): text "ePPS1 %s"; shows .PPS1_emul
  rounded rectangle at (15,275)-(206,326): text "cPPS1 %s"; shows .cPPS1_emul
  rounded rectangle at (15,150)-(206,201): text "dPPS1 %s"; shows .PPS1-.PPS1_emul
  rounded rectangle at (15,215)-(206,266): text "Emul %%  %s"; shows 100-((.PPS1_emul-.p.PPS_table[1])*100)/(.PPS1-.p.PPS_table[1])
group at (895,10)-(1216,371)
  rounded rectangle at (10,210)-(221,263): text "Red temp %s"; shows .Reductor_temp
  rounded rectangle at (10,80)-(221,131): text "HOLD %s"; shows .HOLD_time
  rounded rectangle at (10,140)-(221,195): text "Red press %s"; shows .Reductor_press
  rounded rectangle at (10,20)-(221,71): text "Itemp %s"; shows .Injector_temp
  rounded rectangle at (10,280)-(221,331): text "Tblock %s"; shows .gs16_TempBoard
  rectangle at (230,20)-(306,71): text "%s"; shows .p.Inj_temp_max
  rectangle at (230,80)-(306,131): text "%s"; shows .p.Inj_MAX_hold_time/4
  rectangle at (230,140)-(306,191): text "%s"; shows .p.Min_Reductor_press
  rectangle at (230,210)-(306,261): text "%s"; shows .p.Reductor_temp_work
rounded rectangle at (660,360)-(861,416): text "Speed lim %s"; shows .p.Speed_table[12]
rounded rectangle at (660,430)-(861,486): text "GAS cor %2.2f"; shows Act_control.Gas_Speed_cor
rounded rectangle at (660,495)-(861,551): text "DT cor %2.2f"; shows Act_control.Diesel_Speed_cor
button at (40,270)-(156,316): text "PWM adj"; opens PWM_adjustment
button at (40,90)-(156,136): text "SETUP"; opens SETUP
button at (40,210)-(156,256): text "Check Current"; opens CHECK_CURRENT
button at (35,150)-(156,196): text "Check EGT"; opens CHECK_EGT
button at (40,35)-(156,81): text "Calibration"; opens CALIBRATION
group at (230,25)-(326,401)
  ellipse at (10,93)-(86,157): text "Safety / relay"; alarm colour if .gq_Relay
  ellipse at (10,9)-(86,74): text "BLOCK / ON"; alarm colour if .Flag_ECU_ON
  button at (15,176)-(76,226): text "Manual / ON"; toggles .Flag_ECU_ON_VISU
  ellipse at (15,240)-(76,301): text "SPEED / OK"; alarm colour if Get_RPM_speed.Flag_speed_OK
  rectangle at (15,310)-(81,351): text "%s"; shows .p.Speed_limit
rounded rectangle at (175,520)-(366,576): text "EGT  %s"; shows .EGT
rounded rectangle at (175,590)-(361,646): text "GAS cor %2.2f"; shows Act_control.Gas_EGT_cor
rounded rectangle at (175,655)-(361,711): text "DT cor %2.2f"; shows Act_control.Diesel_EGT_cor
rectangle at (235,435)-(316,486): text "%s"; shows .p.EGT_max
35 more shapes without text or variables
*)

(* Visualisation PWM_ADJUSTMENT
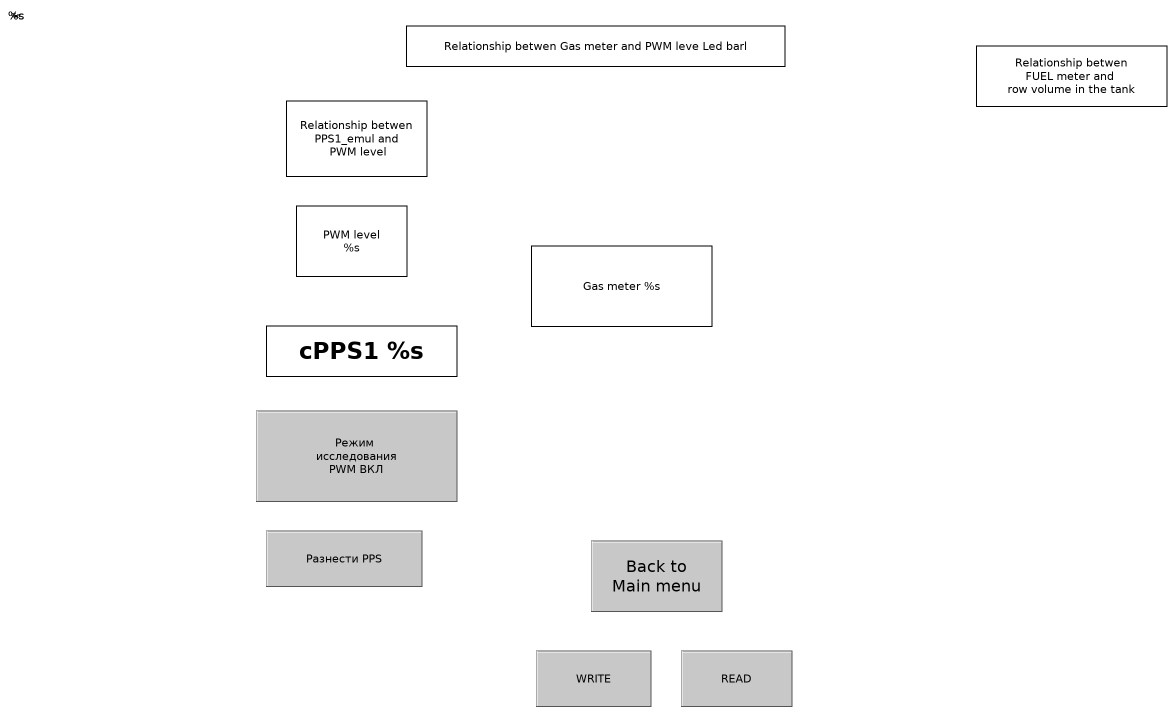
button at (240,395)-(441,486): text "Режим / исследования / PWM ВКЛ"; toggles .Flag_PWM_researh
rounded rectangle at (270,85)-(411,161): text "Relationship betwen / PPS1_emul and / PWM level"
rounded rectangle at (280,190)-(391,261): text "PWM level / %s"; shows Act_control.PPS_PWM; editable
rectangle at (0,0)-(0,0): text "%s"; shows p.PPS1_emul_PWM[INDEX]; editable
rectangle at (0,0)-(0,0): text "%s"; shows p.PPS_table[INDEX]; editable
rounded rectangle at (250,310)-(441,361): text "cPPS1 %s"; shows .cPPS1_emul
button at (575,525)-(706,596): text "Back to / Main menu"; opens PLC_VISU
group at (520,635)-(776,691)
  button at (0,0)-(115,56): text "WRITE"; taps DFPRS_Change_Cal_Table.Write_cal
  button at (145,0)-(256,56): text "READ"; taps DFPRS_Change_Cal_Table.Read_cal
rounded rectangle at (960,30)-(1151,91): text "Relationship betwen / FUEL meter and / row volume in the tank"
rounded rectangle at (390,10)-(769,51): text "Relationship betwen Gas meter and PWM leve Led barl"
rounded rectangle at (515,230)-(696,311): text "Gas meter %s"; shows .Gas_meter
rectangle at (0,0)-(0,0): text "%s"; shows p.LED_BAR_PWM[INDEX]; editable
rectangle at (0,0)-(0,0): text "%s"; shows p.Gas_meter_volume[INDEX]; editable
button at (250,515)-(406,571): text "Разнести PPS"; taps DFPRS_Change_Cal_Table.Flag_PPS_raznoska; runs 222
*)

(* Visualisation SETUP
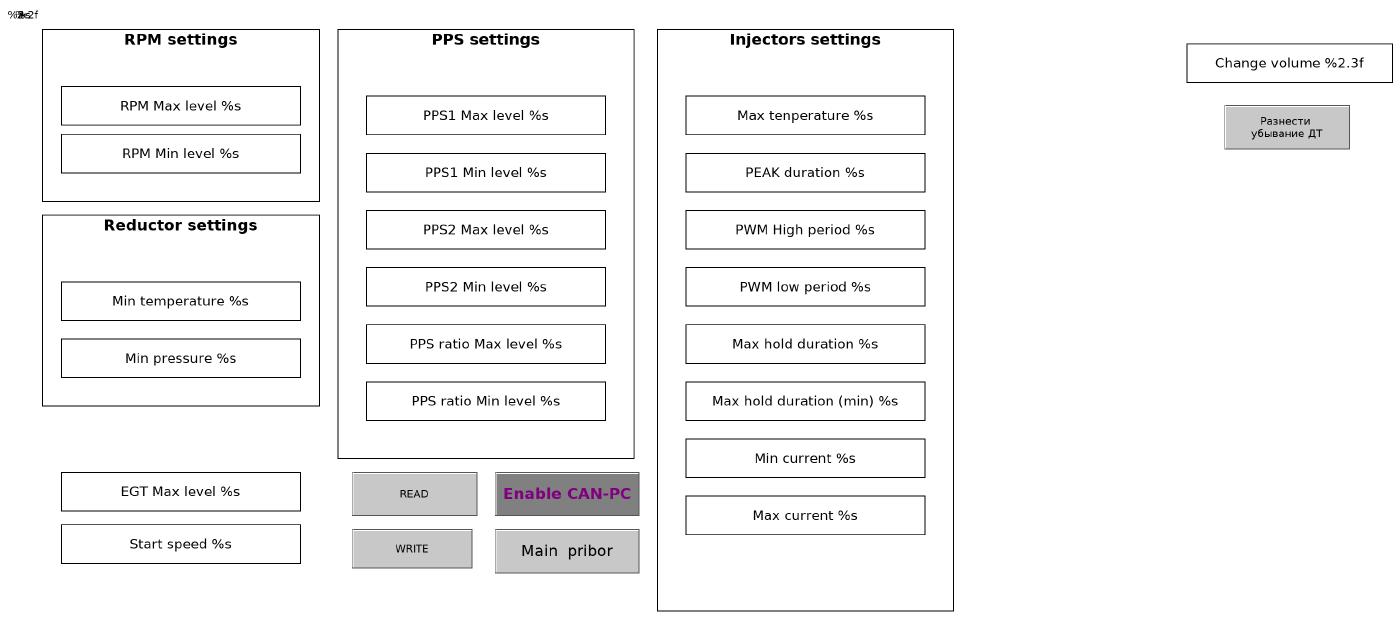
rounded rectangle at (20,210)-(311,411): text "Reductor settings"
rounded rectangle at (20,15)-(311,196): text "RPM settings"
button at (495,480)-(646,526): text "Enable CAN-PC"; toggles .Flag_CAN
rounded rectangle at (40,480)-(291,521): text "EGT Max level %s"; shows .p.EGT_max; editable
button at (345,480)-(476,526): text "READ"; taps DFPRS_Change_Cal_Table.Read_cal
button at (345,540)-(471,581): text "WRITE"; taps DFPRS_Change_Cal_Table.Write_cal
button at (495,540)-(646,586): text "Main  pribor"; opens PLC_VISU
rounded rectangle at (40,75)-(291,116): text "RPM Max level %s"; shows .p.RPM_max; editable
rounded rectangle at (40,125)-(291,166): text "RPM Min level %s"; shows .p.RPM_min; editable
rounded rectangle at (40,280)-(291,321): text "Min temperature %s"; shows .p.Reductor_temp_work; editable
rounded rectangle at (40,340)-(291,381): text "Min pressure %s"; shows .p.Min_Reductor_press; editable
rounded rectangle at (330,15)-(641,466): text "PPS settings"
rounded rectangle at (360,85)-(611,126): text "PPS1 Max level %s"; shows .p.PPS1_max; editable
rounded rectangle at (360,145)-(611,186): text "PPS1 Min level %s"; shows .p.PPS1_min; editable
rounded rectangle at (360,205)-(611,246): text "PPS2 Max level %s"; shows .p.PPS2_max; editable
rounded rectangle at (360,265)-(611,306): text "PPS2 Min level %s"; shows .p.PPS2_min; editable
rounded rectangle at (360,325)-(611,366): text "PPS ratio Max level %s"; shows .p.PPS_ratio_max; editable
rounded rectangle at (360,385)-(611,426): text "PPS ratio Min level %s"; shows .p.PPS_ratio_min; editable
rounded rectangle at (665,15)-(976,626): text "Injectors settings"; tooltip Значения настроек для инжекторов надо менять очень осторожно. И хорошо представлять себя последствия.
rounded rectangle at (695,325)-(946,366): text "Max hold duration %s"; shows .p.Inj_MAX_hold_time; tooltip Абсолютное ограничение максимальной длительности тока удержания. Задается в циклах по 250 мкс. HOLD 1 мс =4*250 мкс; editable
rounded rectangle at (695,385)-(946,426): text "Max hold duration (min) %s"; shows .p.Inj_MAX_hold_time_min; tooltip Ограничение максимальной длительности тока удержания для первых трех значений RPM и Turbo Задается в циклах по 250 мкс. HOLD 1 мс =4*250 мкс; editable
rounded rectangle at (695,265)-(946,306): text "PWM low period %s"; shows .p.Inj_Low_period; tooltip Задание скважности PWM форсунок ( соотношение кол-ва ЦИКЛОВ низкого сигнала к одному ВЫСОКОМУ циклу ), подбирается имперически по условию соблюдения уровня холдового тока на форсунке; editable
rounded rectangle at (695,205)-(946,246): text "PWM High period %s"; shows .p.Inj_High_period; tooltip Задание скважности PWM форсунок ( соотношение кол-ва ЦИКЛОВ низкого сигнала к одному ВЫСОКОМУ циклу ), подбирается имперически по условию соблюдения уровня холдового тока на форсунке; editable
rounded rectangle at (695,145)-(946,186): text "PEAK duration %s"; shows .p.Inj_peak_curent_cycle; tooltip Количество циклов по 250 мкс для генерирования пикового импульса открытия форсунки; editable
rounded rectangle at (695,85)-(946,126): text "Max tenperature %s"; shows .p.Inj_temp_max; tooltip Максимальный ток в микроамперах, протекающий через терморезистор на рейке; editable
rounded rectangle at (695,445)-(946,486): text "Min current %s"; shows .p.Min_inj_current; tooltip Минимальный длительный ток через форсунки; editable
rounded rectangle at (695,505)-(946,546): text "Max current %s"; shows .p.Max_inj_current; tooltip Максимальный длительный ток через форсунки; editable
rounded rectangle at (40,535)-(291,576): text "Start speed %s"; shows .p.Speed_limit; editable
rectangle at (0,0)-(0,0): text "%s"; shows p.EGT_table[INDEX]; editable
rectangle at (0,0)-(0,0): text "%s"; shows p.GAS_EGT_table[INDEX]; editable
rectangle at (0,0)-(0,0): text "%s"; shows p.DIESEL_EGT_table[INDEX]; editable
rectangle at (0,0)-(0,0): text "%s"; shows p.Load_table[INDEX]; editable
rectangle at (0,0)-(0,0): text "%s"; shows p.GAS_Load_table[INDEX]; editable
rectangle at (0,0)-(0,0): text "%s"; shows p.DIESEL_Load_table[INDEX]; editable
rectangle at (0,0)-(0,0): text "%s"; shows p.Speed_table[INDEX]; editable
rectangle at (0,0)-(0,0): text "%s"; shows p.GAS_Speed_table[INDEX]; editable
rectangle at (0,0)-(0,0): text "%2.2f"; shows p.DIESEL_Speed_table[INDEX]; editable
rounded rectangle at (1220,30)-(1436,71): text "Change volume %2.3f"; shows DFPRS_Change_Cal_Table.Speed_limit_step; tooltip Максимальный ток в микроамперах, протекающий через терморезистор на рейке; editable
button at (1260,95)-(1391,141): text "Разнести / убывание ДТ"; taps DFPRS_Change_Cal_Table.Flag_speed_limit_raznoska
*)
